// TIA Portal V20 export
TYPE "zm_Cycletype"
// stored: Access Published
   STRUCT
      EndOfCycle : Bool;
      DryRun : Bool;
      RunOut : Bool;
      GaugeRnRtype1 : Bool;
      reserved : Bool;
      GaugeRnRtype3 : Bool;
      bypass : Bool;
      Reserved_0 : Bool;
      Reserved_1 : Bool;
      Reserved_2 : Bool;
      Reserved_3 : Bool;
      Reserved_4 : Bool;
      Reserved_5 : Bool;
      Reserved_6 : Bool;
      Reserved_7 : Bool;
      Reserved_8 : Bool;
      Reserved_9 : Bool;
      Reserved_10 : Bool;
      Reserved_11 : Bool;
      Reserved_12 : Bool;
      Reserved_13 : Bool;
      Reserved_14 : Bool;
      Reserved_15 : Bool;
      Reserved_16 : Bool;
      Reserved_17 : Bool;
      Reserved_18 : Bool;
      Reserved_19 : Bool;
      Reserved_20 : Bool;
      Reserved_21 : Bool;
      Reserved_22 : Bool;
      Reserved_23 : Bool;
      Reserved_24 : Bool;
   END_STRUCT;
END_TYPE
